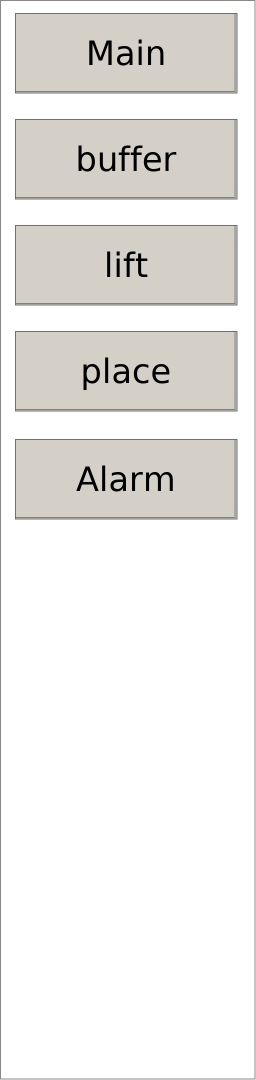
VISUALIZATION Menu  // 256x1080
    Button (15,119 222x80), "buffer", colour toggle: G_HMI.iMainFrame =1
        p573394764: 16#FF00FF00
        OnMouseDown: execute { G_HMI.iMainFrame	:= 1; }
    Button (15,225 222x80), "lift", colour toggle: G_HMI.iMainFrame =2
        p573394764: 16#FF00FF00
        OnMouseDown: execute { G_HMI.iMainFrame	:= 2; }
    Button (15,331 222x80), "place", colour toggle: G_HMI.iMainFrame =3
        p573394764: 16#FF00FF00
        OnMouseDown: execute { G_HMI.iMainFrame	:= 3; }
    Button (15,13 222x80), "Main", colour toggle: G_HMI.iMainFrame =0
        p573394764: 16#FF00FF00
        OnMouseDown: execute { G_HMI.iMainFrame	:= 0; }
    Button (15,439 222x80), "Alarm", colour toggle: G_HMI.iMainFrame =4
        p573394764: 16#FF00FF00
        OnMouseDown: execute { G_HMI.iMainFrame	:= 4; }
END_VISUALIZATION

(* stored: Version 1.1.0.1, ProductVersion 3.1.4024.12
   Visu Menu: Id {2c1cc129-5e67-4f8a-b890-3aee9edbaf72} *)
